// TIA Portal V17 export
// export: Created 2025-06-26T06:49:16.3931886Z, ExportSetting WithDefaults, DisplayName Totally Integrated Automation Portal, DisplayVersion V17 Update 8, DisplayName TIA Portal Openness, DisplayVersion V17 Update 8, DisplayName TIA Portal Version Control Interface, DisplayVersion V17, DisplayName STEP 7 Professional, DisplayVersion V17 Update 8, DisplayName STEP 7 Safety, DisplayVersion V17 Update 6, DisplayName WinCC Advanced, DisplayVersion V17 Update 8
FUNCTION_BLOCK "fbHMIEvent"   // FB39, FBD
{ S7_Optimized_Access := 'TRUE' }
VERSION : 0.1
// stored: AutoNumber true, IsIECCheckEnabled false, IsRetainMemResEnabled false, MemoryReserve 0, SetENOAutomatically false, UDAEnableTagReadback false
   VAR_INPUT
      bInput : Bool;
      bAckAll : Bool;
      bEnable : Bool;
   END_VAR
   VAR_IN_OUT
      sTag : "stEvent";
   END_VAR
   VAR
      Event : "fbEvent";
   END_VAR
BEGIN

REGION Network 1
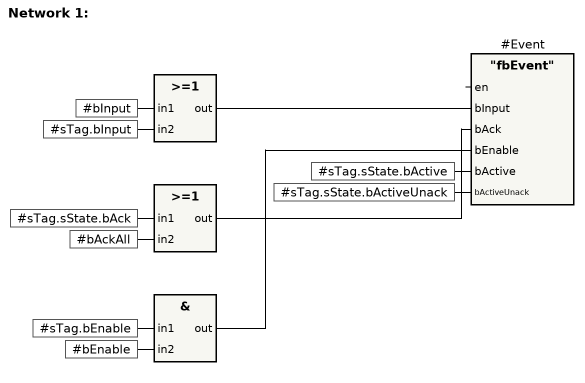
   #Event(bInput := #bInput OR #sTag.bInput,   // "fbEvent"
          bAck := #sTag.sState.bAck OR #bAckAll,
          bEnable := #sTag.bEnable AND #bEnable,
          bActive := #sTag.sState.bActive,
          bActiveUnack := #sTag.sState.bActiveUnack);
END_REGION
END_FUNCTION_BLOCK
